FUNCTION PwmSignal : REAL
VAR_INPUT
	ymin:				REAL; 	//Minimalwert
	ymax:				REAL; 	//Maximalwert
	w:					REAL; 	//Kreisfrequenz
	yoff:				REAL; 	//yoffset
	PWM:				REAL;	//PWM 0.0 ... 1.0%
	t : 				REAL;	//Zeit
END_VAR
VAR
	tempTime:			REAL;
END_VAR

tempTime := LMOD(lr_Value:=t,lr_Arg:=(2*PI)/w)/((2*PI)/w);

IF(PWM = 1) THEN
	PwmSignal := ymax + yoff;
	RETURN;
END_IF
IF(tempTime <= (1-PWM)) THEN
	PwmSignal := ymin + yoff;
	RETURN;
ELSE
	PwmSignal := ymax + yoff;
	RETURN;
END_IF

END_FUNCTION

(* stored: Version 1.1.0.1, ProductVersion 3.1.4024.13
   POU PwmSignal: Id {302c83ed-f0e7-4793-b1d8-1a1b3f61c62f}, SpecialFunc None *)
